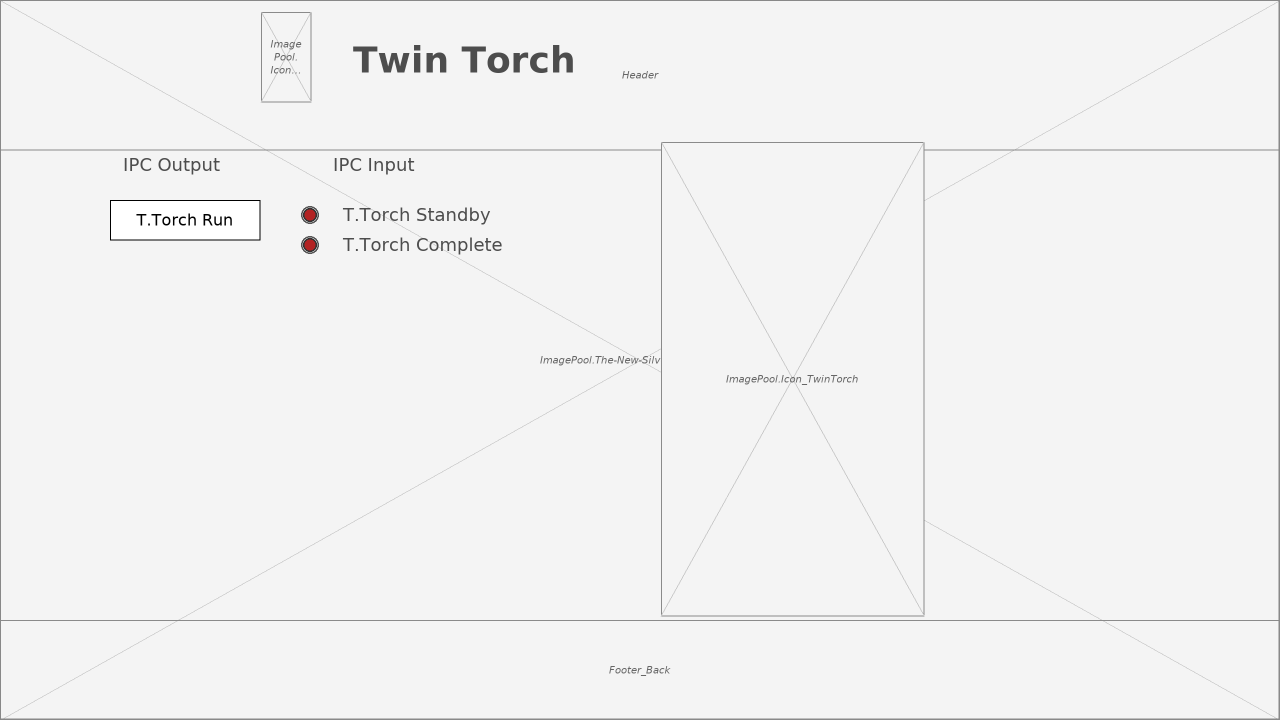
VISUALIZATION PAGE_TTorch  // 1280x720
    Image (0,0 1280x720), image: ImagePool.The-New-Silver-Backgrounds
    Frame (0,620 1280x100)
        shows Footer_Back()
    Frame (0,0 1280x150)
        shows Header()
    Label (350,40 300x40), "Twin Torch"
    Label (120,150 150x30), "IPC Output"
    RoundedRectangle (110,200 150x40), "T.Torch Run"
        toggle GVL.TTorch_Run
    Label (330,150 150x30), "IPC Input"
    Label (340,200 170x30), "T.Torch Standby"
    Lamp1 (300,205 20x20), variable: GVL.TTorch_Standy, style: Lamp-Lamp1-Red
    Label (340,230 170x30), "T.Torch Complete"
    Lamp1 (300,235 20x20), variable: GVL.TTorch_Complete, style: Lamp-Lamp1-Red
    Image (261,12 50x90), image: ImagePool.Icon_TwinTorch
    Image (661,142 263x474), image: ImagePool.Icon_TwinTorch
END_VISUALIZATION

(* stored: Version 1.1.0.1, ProductVersion 3.1.4024.12
   Visu PAGE_TTorch: Id {a75d410e-c234-4b25-b13d-2c3817f71ee4} *)
